PROGRAM MAIN
VAR
END_VAR

//Main POU

END_PROGRAM

(* stored: Version 1.1.0.1, ProductVersion 3.1.4024.12
   POU MAIN: Id {02fb42c5-c1a2-4e52-b2e2-9a90d275cfb1}, SpecialFunc None *)
